PROGRAM Read_Pressure
VAR
	EL3052_Lead_Bit AT %I* : INT;
	EL3052_Rear_Bit AT %I* : INT;
	
	Pressure_Lead		: REAL;
	Pressure_Rear		: REAL;
	Threshold			: REAL := 180;
	
	Overpressure_Lead	: BOOL;
	Overpressure_Rear	: BOOL;
	
END_VAR

(* read pressure *)
IF GVL.Lead_Trailer_State = 8 OR GVL.Lead_Trailer_State = 17416 THEN
	Pressure_Lead 	:= (INT_TO_REAL(EL3052_Lead_Bit)/32767) * 160;
ELSE
	Pressure_Lead 	:= 0;	
END_IF

IF GVL.Rear_Trailer_State = 8 THEN
	Pressure_Rear 	:= (INT_TO_REAL(EL3052_Rear_Bit)/32767) * 160;
ELSE
	Pressure_Rear 	:= 0;
END_IF

(* check for overpressure *)
IF Pressure_Lead > Threshold THEN
	Overpressure_Lead := TRUE;
ELSE
	Overpressure_Lead := FALSE;
END_IF

IF Pressure_Rear > Threshold THEN
	Overpressure_Rear := TRUE;
ELSE
	Overpressure_Rear := FALSE;
END_IF

(* only read over pressure event once during dump cycle *)

END_PROGRAM

(* stored: Version 1.1.0.1, ProductVersion 3.1.4024.6
   POU Read_Pressure: Id {4da627ee-194f-436f-bf88-e2e5c518b461}, SpecialFunc None *)
